(* IEC 61131-3 sources: crb-codesys/retrieval/output/codesys_repo/开放式双周卷绕机编程开发实训 copy/FUN, 8 files *)

(* ---- CheckF.st ---- *)
FUNCTION_BLOCK CheckF
VAR_INPUT
	lM	:	LREAL;
	lL	:	LREAL;
	lH	:	LREAL;
END_VAR
VAR_OUTPUT
	lF	:	LREAL;
END_VAR
VAR
END_VAR

IF lH<>0 THEN
	lF:=9.8*lM/(2*COS(ATAN(lL/lH)));
END_IF

(* ---- SeekHome.st ---- *)
FUNCTION_BLOCK SeekHome
VAR_IN_OUT
	_Axis	:	AXIS_REF_SM3;
END_VAR
VAR_INPUT
	_xHome	:	BOOL;
	_xAbort	:	BOOL;
	_nHomeMode	:	HomeMode;
	_fFastHomeVel	:	LREAL;
	_fSlowHomeVel	:	LREAL;
	_fHomeAcc		:	LREAL;
	_fHomeDec		:	LREAL;
	_fHomePos		:	LREAL;
	_xReferenceSwitch	:	BOOL;//typically is true
	_nDirection	:	MC_DIRECTION;
	_xIndexPulse	:	BOOL;
END_VAR
VAR_OUTPUT
	_xBusy	:	BOOL;
	_xDone	:	BOOL;
	_xErr	:	BOOL;
	_iErrId	:	DINT;
END_VAR
VAR
	_fbMoveVel	:	MC_MoveVelocity;
	_fbMoveAbs	:	MC_MoveAbsolute;
	_fbHalt		:	MC_Halt;
	_fbSetPos	:	MC_SetPosition;
	_fbRtrig		:	R_TRIG;
	_fbFtrig		:	F_TRIG;
	_nBDirection	:	MC_DIRECTION;
	_fTempPos		:	LREAL;
	_nState		:	USINT;
	fbRtrig	:	R_TRIG;
END_VAR

//check left / arrive the ReferenceSwitch
_fbRtrig(CLK := _xReferenceSwitch);
_fbFtrig(CLK := _xReferenceSwitch);
fbRtrig(CLK := _xHome);

IF NOT _xHome THEN
	_fbMoveVel(Axis := _Axis,Execute := FALSE);
	_fbMoveAbs(Axis := _Axis,Execute := FALSE);
	_fbHalt(Axis := _Axis,Execute := FALSE);
	_fbSetPos(Axis := _Axis,Execute := FALSE);
	_xDone := FALSE;
	_xErr := FALSE;
END_IF

CASE _nState OF
	0:
		IF fbRtrig.Q THEN
			_xBusy := TRUE;
			_xDone := FALSE;
			_xErr := FALSE;
			_iErrId := 0;

			CASE _nDirection OF //cal which is the invert direction
				MC_DIRECTION.positive:
					_nBDirection := MC_DIRECTION.negative;
				MC_DIRECTION.negative:
					_nBDirection := MC_DIRECTION.positive;
				ELSE
					_xErr := TRUE;
			END_CASE

			CASE _nHomeMode OF
				HomeMode.FAST_ZERO:
					_fTempPos := 0;
					_nState := 21;
				HomeMode.FAST_BSLOW_STOP_S:
					_nState := 1;
				HomeMode.FAST_SLOW_STOP_S:
					_nState := 11;
				HomeMode.FAST_BSLOW_I_STOP_S:
					_nState := 31;
				HomeMode.FAST_SLOW_I_STOP_S:
					_nState := 41;
			END_CASE
		END_IF
	50:
		_fbMoveAbs(Execute := TRUE,Axis := _Axis,Position := _fTempPos,Velocity := _fSlowHomeVel,Acceleration := _fHomeAcc,Deceleration := _fHomeDec);
		IF _fbMoveAbs.Done THEN
			_fbMoveAbs(Execute := FALSE,Axis := _Axis);
			_nState := 100;
		END_IF
		IF _fbMoveAbs.Error THEN//meet error
			_nState := 200;
			_iErrId := _fbMoveAbs.ErrorID;
		END_IF
	100:
		_fbSetPos(Execute := TRUE,Axis := _Axis,Position := _fHomePos,Mode := FALSE);//set absolute position
		IF _fbSetPos.Done THEN
			_fbSetPos(Execute := FALSE,Axis := _Axis);
			_xDone := TRUE;
			_xBusy := FALSE;
			_nState := 0;
		END_IF
		IF _fbSetPos.Error THEN//meet error
			_iErrId := _fbSetPos.ErrorID;
			_nState := 200;
		END_IF
	200:
		_xErr := TRUE;
		_xBusy := FALSE;
		_nState := 0;
END_CASE

FAST_ZERO();
FAST_BSLOW_STOP_S();
FAST_SLOW_STOP_S();
FAST_BSLOW_I_STOP_S();
FAST_SLOW_I_STOP_S();

(* ---- StaDisplay.st ---- *)
FUNCTION_BLOCK StaDisplay
VAR_INPUT
	iStatus :	INT;
END_VAR
VAR_OUTPUT
	Y1,Y2,Y3,Y4,Y5,Y6	:	BOOL;
END_VAR
VAR
END_VAR

CASE iStatus OF
	2,3,4,5,6,7,8,9,10,221,222:
	Y5:=FALSE;
	Y6:=TRUE;
	Y1:=TRUE;
	Y2:=FALSE;
	Y3:=FALSE;
	Y4:=FALSE;
	11,12:
	Y5:=FALSE;
	Y6:=TRUE;
	Y1:=FALSE;
	Y2:=TRUE;
	Y3:=FALSE;
	Y4:=FALSE;
	13,14,15,16,17,18,19,20,21,22:
	Y5:=TRUE;
	Y6:=FALSE;
	Y1:=FALSE;
	Y2:=FALSE;
	Y3:=TRUE;
	Y4:=FALSE;
	23,24:
	Y5:=TRUE;
	Y6:=FALSE;
	Y1:=FALSE;
	Y2:=FALSE;
	Y3:=FALSE;
	Y4:=TRUE;
	ELSE
	Y5:=TRUE;
	Y6:=TRUE;
	Y1:=FALSE;
	Y2:=FALSE;
	Y3:=FALSE;
	Y4:=FALSE;
END_CASE

(* ---- SeekHome_FAST_BSLOW_I_STOP_S.st ---- *)
METHOD FAST_BSLOW_I_STOP_S
VAR_IN_OUT
	_Axis	:	AXIS_REF_SM3;
END_VAR
VAR_INPUT
	_xHome	:	BOOL;
	_xAbort	:	BOOL;
	_nHomeMode	:	HomeMode;
	_fFastHomeVel	:	LREAL;
	_fSlowHomeVel	:	LREAL;
	_fHomeAcc		:	LREAL;
	_fHomeDec		:	LREAL;
	_fHomePos		:	LREAL;
	_xReferenceSwitch	:	BOOL;//typically is true
	_nDirection	:	MC_DIRECTION;
	_xIndexPulse	:	BOOL;
END_VAR
VAR_OUTPUT
	_xBusy	:	BOOL;
	_xDone	:	BOOL;
	_xErr	:	BOOL;
	_iErrId	:	DINT;
END_VAR
VAR
	_fbMoveVel	:	MC_MoveVelocity;
	_fbMoveAbs	:	MC_MoveAbsolute;
	_fbHalt		:	MC_Halt;
	_fbSetPos	:	MC_SetPosition;
	_fbRtrig		:	R_TRIG;
	_fbFtrig		:	F_TRIG;
	_nBDirection	:	MC_DIRECTION;
	_fTempPos		:	LREAL;
	_nState		:	USINT;
	fbRtrig	:	R_TRIG;
END_VAR

CASE _nState OF
	31:
		IF _xReferenceSwitch THEN
			_nState := 33;//out of ReferenceSwitch
		ELSE
			_nState :=32;//in the ReferenceSwitch
		END_IF

		_fbMoveAbs(Execute := FALSE,Axis := _Axis);
		_fbSetPos(Execute := FALSE,Axis := _Axis);
		_fbMoveVel(Execute := FALSE,Axis := _Axis);
	32://move out of the ReferenceSwitch
		_fbMoveVel(Execute := TRUE,Axis := _Axis,Velocity := _fSlowHomeVel,Acceleration := _fHomeAcc,Deceleration := _fHomeDec,Direction := _nBDirection);
		IF _fbRtrig.Q THEN//left the ReferenceSwitch
			_nState := 34;
		END_IF
		IF _fbMoveVel.Error THEN//meet error
			_iErrId := _fbMoveVel.ErrorID;
			_fbMoveVel(Execute := FALSE,Axis := _Axis);
			_nState := 200;
		END_IF
	33://move to ReferenceSwitch
		_fbMoveVel(Execute := TRUE,Axis := _Axis,Velocity := _fFastHomeVel,Acceleration := _fHomeAcc,Deceleration := _fHomeDec,Direction := _nDirection);
		IF _fbFtrig.Q THEN//arrive the ReferenceSwitch
			_fbMoveVel(Execute := FALSE,Axis := _Axis);
			_nState := 32;
		END_IF
		IF _fbMoveVel.Error THEN//meet error
			_iErrId := _fbMoveVel.ErrorID;
			_fbMoveVel(Execute := FALSE,Axis := _Axis);
			_nState := 200;
		END_IF
	34:
		_fbMoveVel(Execute := TRUE,Axis := _Axis,Velocity := _fSlowHomeVel,Acceleration := _fHomeAcc,Deceleration := _fHomeDec,Direction := _nBDirection);
		IF _xIndexPulse THEN//left the ReferenceSwitch
			_fTempPos := _Axis.fActPosition;//save the position
			_fbMoveVel(Execute := FALSE,Axis := _Axis);
			_nState := 50;
		END_IF
		IF _fbMoveVel.Error THEN//meet error
			_iErrId := _fbMoveVel.ErrorID;
			_fbMoveVel(Execute := FALSE,Axis := _Axis);
			_nState := 200;
		END_IF
END_CASE

(* ---- SeekHome_FAST_BSLOW_STOP_S.st ---- *)
METHOD FAST_BSLOW_STOP_S
VAR_IN_OUT
	_Axis	:	AXIS_REF_SM3;
END_VAR
VAR_INPUT
	_xHome	:	BOOL;
	_xAbort	:	BOOL;
	_nHomeMode	:	HomeMode;
	_fFastHomeVel	:	LREAL;
	_fSlowHomeVel	:	LREAL;
	_fHomeAcc		:	LREAL;
	_fHomeDec		:	LREAL;
	_fHomePos		:	LREAL;
	_xReferenceSwitch	:	BOOL;//typically is true
	_nDirection	:	MC_DIRECTION;
	_xIndexPulse	:	BOOL;
END_VAR
VAR_OUTPUT
	_xBusy	:	BOOL;
	_xDone	:	BOOL;
	_xErr	:	BOOL;
	_iErrId	:	DINT;
END_VAR
VAR
	_fbMoveVel	:	MC_MoveVelocity;
	_fbMoveAbs	:	MC_MoveAbsolute;
	_fbHalt		:	MC_Halt;
	_fbSetPos	:	MC_SetPosition;
	_fbRtrig		:	R_TRIG;
	_fbFtrig		:	F_TRIG;
	_nBDirection	:	MC_DIRECTION;
	_fTempPos		:	LREAL;
	_nState		:	USINT;
	fbRtrig	:	R_TRIG;
END_VAR

CASE _nState OF
	1:
		IF _xReferenceSwitch THEN
			_nState := 2;//out of ReferenceSwitch
		ELSE
			_nState :=3;//in the ReferenceSwitch
		END_IF

		_fbMoveAbs(Execute := FALSE,Axis := _Axis);
		_fbSetPos(Execute := FALSE,Axis := _Axis);
		_fbMoveVel(Execute := FALSE,Axis := _Axis);
	2://move out of the ReferenceSwitch
		_fbMoveVel(Execute := TRUE,Axis := _Axis,Velocity := _fSlowHomeVel,Acceleration := _fHomeAcc,Deceleration := _fHomeDec,Direction := _nBDirection);
		IF _fbFtrig.Q THEN//left the ReferenceSwitch
			_fTempPos := _Axis.fActPosition;//save the position
			_fbMoveVel(Execute := FALSE,Axis := _Axis);
			_nState := 50;
		END_IF
		IF _fbMoveVel.Error THEN//meet error
			_iErrId := _fbMoveVel.ErrorID;
			_fbMoveVel(Execute := FALSE,Axis := _Axis);
			_nState := 200;
		END_IF

	3://move to ReferenceSwitch
		_fbMoveVel(Execute := TRUE,Axis := _Axis,Velocity := _fFastHomeVel,Acceleration := _fHomeAcc,Deceleration := _fHomeDec,Direction := _nDirection);
		IF _fbRtrig.Q THEN//arrive the ReferenceSwitch
			_fbMoveVel(Execute := FALSE,Axis := _Axis);
			_nState := 2;
		END_IF
		IF _fbMoveVel.Error THEN//meet error
			_iErrId := _fbMoveVel.ErrorID;
			_fbMoveVel(Execute := FALSE,Axis := _Axis);
			_nState := 200;
		END_IF
END_CASE

(* ---- SeekHome_FAST_SLOW_I_STOP_S.st ---- *)
METHOD FAST_SLOW_I_STOP_S
VAR_IN_OUT
	_Axis	:	AXIS_REF_SM3;
END_VAR
VAR_INPUT
	_xHome	:	BOOL;
	_xAbort	:	BOOL;
	_nHomeMode	:	HomeMode;
	_fFastHomeVel	:	LREAL;
	_fSlowHomeVel	:	LREAL;
	_fHomeAcc		:	LREAL;
	_fHomeDec		:	LREAL;
	_fHomePos		:	LREAL;
	_xReferenceSwitch	:	BOOL;//typically is true
	_nDirection	:	MC_DIRECTION;
	_xIndexPulse	:	BOOL;
END_VAR
VAR_OUTPUT
	_xBusy	:	BOOL;
	_xDone	:	BOOL;
	_xErr	:	BOOL;
	_iErrId	:	DINT;
END_VAR
VAR
	_fbMoveVel	:	MC_MoveVelocity;
	_fbMoveAbs	:	MC_MoveAbsolute;
	_fbHalt		:	MC_Halt;
	_fbSetPos	:	MC_SetPosition;
	_fbRtrig		:	R_TRIG;
	_fbFtrig		:	F_TRIG;
	_nBDirection	:	MC_DIRECTION;
	_fTempPos		:	LREAL;
	_nState		:	USINT;
	fbRtrig	:	R_TRIG;
END_VAR

CASE _nState OF
	41:
		IF _xReferenceSwitch THEN
			_nState := 43;//out of ReferenceSwitch
		ELSE
			_nState := 42;//in the ReferenceSwitch
		END_IF

		_fbMoveAbs(Execute := FALSE,Axis := _Axis);
		_fbSetPos(Execute := FALSE,Axis := _Axis);
		_fbMoveVel(Execute := FALSE,Axis := _Axis);
	42://move out of the ReferenceSwitch
		_fbMoveVel(Execute := TRUE,Axis := _Axis,Velocity := _fSlowHomeVel,Acceleration := _fHomeAcc,Deceleration := _fHomeDec,Direction := _nDirection);
		IF _fbRtrig.Q THEN//left the ReferenceSwitch
			_nState := 44;
		END_IF
		IF _fbMoveVel.Error THEN//meet error
			_iErrId := _fbMoveVel.ErrorID;
			_fbMoveVel(Execute := FALSE,Axis := _Axis);
			_nState := 200;
		END_IF
	43://move to ReferenceSwitch
		_fbMoveVel(Execute := TRUE,Axis := _Axis,Velocity := _fFastHomeVel,Acceleration := _fHomeAcc,Deceleration := _fHomeDec,Direction := _nDirection);
		IF _fbFtrig.Q THEN//arrive the ReferenceSwitch
			_fbMoveVel(Execute := FALSE,Axis := _Axis);
			_nState := 42;
		END_IF
		IF _fbMoveVel.Error THEN//meet error
			_iErrId := _fbMoveVel.ErrorID;
			_fbMoveVel(Execute := FALSE,Axis := _Axis);
			_nState := 200;
		END_IF
	44:
		_fbMoveVel(Execute := TRUE,Axis := _Axis,Velocity := _fSlowHomeVel,Acceleration := _fHomeAcc,Deceleration := _fHomeDec,Direction := _nDirection);
		IF _xIndexPulse THEN//left the ReferenceSwitch
			_fTempPos := _Axis.fActPosition;//save the position
			_fbMoveVel(Execute := FALSE,Axis := _Axis);
			_nState := 50;
		END_IF
		IF _fbMoveVel.Error THEN//meet error
			_iErrId := _fbMoveVel.ErrorID;
			_fbMoveVel(Execute := FALSE,Axis := _Axis);
			_nState := 200;
		END_IF
END_CASE

(* ---- SeekHome_FAST_SLOW_STOP_S.st ---- *)
METHOD FAST_SLOW_STOP_S
VAR_IN_OUT
	_Axis	:	AXIS_REF_SM3;
END_VAR
VAR_INPUT
	_xHome	:	BOOL;
	_xAbort	:	BOOL;
	_nHomeMode	:	HomeMode;
	_fFastHomeVel	:	LREAL;
	_fSlowHomeVel	:	LREAL;
	_fHomeAcc		:	LREAL;
	_fHomeDec		:	LREAL;
	_fHomePos		:	LREAL;
	_xReferenceSwitch	:	BOOL;//typically is true
	_nDirection	:	MC_DIRECTION;
	_xIndexPulse	:	BOOL;
END_VAR
VAR_OUTPUT
	_xBusy	:	BOOL;
	_xDone	:	BOOL;
	_xErr	:	BOOL;
	_iErrId	:	DINT;
END_VAR
VAR
	_fbMoveVel	:	MC_MoveVelocity;
	_fbMoveAbs	:	MC_MoveAbsolute;
	_fbHalt		:	MC_Halt;
	_fbSetPos	:	MC_SetPosition;
	_fbRtrig		:	R_TRIG;
	_fbFtrig		:	F_TRIG;
	_nBDirection	:	MC_DIRECTION;
	_fTempPos		:	LREAL;
	_nState		:	USINT;
	fbRtrig	:	R_TRIG;
END_VAR

CASE _nState OF
	11:
		IF _xReferenceSwitch THEN
			_nState := 13;//out of ReferenceSwitch
		ELSE
			_nState :=12;//in the ReferenceSwitch
		END_IF

		_fbMoveAbs(Execute := FALSE,Axis := _Axis);
		_fbSetPos(Execute := FALSE,Axis := _Axis);
		_fbMoveVel(Execute := FALSE,Axis := _Axis);
	12://move out of the ReferenceSwitch
		_fbMoveVel(Execute := TRUE,Axis := _Axis,Velocity := _fSlowHomeVel,Acceleration := _fHomeAcc,Deceleration := _fHomeDec,Direction := _nDirection);
		IF _fbRtrig.Q THEN//left the ReferenceSwitch
			_fTempPos := _Axis.fActPosition;//save the position
			_fbMoveVel(Execute := FALSE,Axis := _Axis);
			_nState := 50;
		END_IF
		IF _fbMoveVel.Error THEN//meet error
			_iErrId := _fbMoveVel.ErrorID;
			_fbMoveVel(Execute := FALSE,Axis := _Axis);
			_nState := 200;
		END_IF
	13://move to ReferenceSwitch
		_fbMoveVel(Execute := TRUE,Axis := _Axis,Velocity := _fFastHomeVel,Acceleration := _fHomeAcc,Deceleration := _fHomeDec,Direction := _nDirection);
		IF _fbFtrig.Q THEN//arrive the ReferenceSwitch
			_fbMoveVel(Execute := FALSE,Axis := _Axis);
			_nState := 12;
		END_IF
		IF _fbMoveVel.Error THEN//meet error
			_iErrId := _fbMoveVel.ErrorID;
			_fbMoveVel(Execute := FALSE,Axis := _Axis);
			_nState := 200;
		END_IF
	50:
		_fbMoveAbs(Execute := TRUE,Axis := _Axis,Position := _fTempPos,Velocity := _fSlowHomeVel,Acceleration := _fHomeAcc,Deceleration := _fHomeDec);
		IF _fbMoveAbs.Done THEN
			_fbMoveAbs(Execute := FALSE,Axis := _Axis);
			_nState := 100;
		END_IF
		IF _fbMoveAbs.Error THEN//meet error
			_nState := 200;
			_iErrId := _fbMoveAbs.ErrorID;
		END_IF
	100:
		_fbSetPos(Execute := TRUE,Axis := _Axis,Position := _fHomePos,Mode := FALSE);//set absolute position
		IF _fbSetPos.Done THEN
			_fbSetPos(Execute := FALSE,Axis := _Axis);
			_xDone := TRUE;
			_xBusy := FALSE;
			_nState := 0;
		END_IF
		IF _fbSetPos.Error THEN//meet error
			_iErrId := _fbSetPos.ErrorID;
			_nState := 200;
		END_IF
	200:
		_xErr := TRUE;
		_xBusy := FALSE;
		_nState := 0;
END_CASE

(* ---- SeekHome_FAST_ZERO.st ---- *)
METHOD FAST_ZERO
VAR_IN_OUT
	_Axis	:	AXIS_REF_SM3;
END_VAR
VAR_INPUT
	_xHome	:	BOOL;
	_xAbort	:	BOOL;
	_nHomeMode	:	HomeMode;
	_fFastHomeVel	:	LREAL;
	_fSlowHomeVel	:	LREAL;
	_fHomeAcc		:	LREAL;
	_fHomeDec		:	LREAL;
	_fHomePos		:	LREAL;
	_xReferenceSwitch	:	BOOL;//typically is true
	_nDirection	:	MC_DIRECTION;
	_xIndexPulse	:	BOOL;
END_VAR
VAR_OUTPUT
	_xBusy	:	BOOL;
	_xDone	:	BOOL;
	_xErr	:	BOOL;
	_iErrId	:	DINT;
END_VAR
VAR
	_fbMoveVel	:	MC_MoveVelocity;
	_fbMoveAbs	:	MC_MoveAbsolute;
	_fbHalt		:	MC_Halt;
	_fbSetPos	:	MC_SetPosition;
	_fbRtrig		:	R_TRIG;
	_fbFtrig		:	F_TRIG;
	_nBDirection	:	MC_DIRECTION;
	_fTempPos		:	LREAL;
	_nState		:	USINT;
	fbRtrig	:	R_TRIG;
END_VAR

CASE _nState OF
	21:
		_fbMoveAbs(Execute := TRUE,Axis := _Axis,Position := _fTempPos,Velocity := _fFastHomeVel,Acceleration := _fHomeAcc,Deceleration := _fHomeDec);
		IF _fbMoveAbs.Done THEN
			_fbMoveAbs(Execute := FALSE,Axis := _Axis);
			_nState := 100;
		END_IF
		IF _fbMoveAbs.Error THEN//meet error
			_nState := 200;
			_iErrId := _fbMoveAbs.ErrorID;
		END_IF
END_CASE
